TYPE E_TcMatSimDataAreaType_1 :
(
	NotSpecified := 0,
	Standard,
	InputSrc,
	InputDst,
	OutputSrc,
	OutputDst,
	InternalDa,
	MArea,
	RetainDa
);
END_TYPE

(* stored: Version 1.1.0.1, ProductVersion 3.1.4020.12
   DUT E_TcMatSimDataAreaType_1: Id {5adc1d66-c048-497c-8757-9c904d8f5dac} *)
